// Mitsubishi GX Works2 project: FRA 451 Class Project NEW   PLC: FX3G

PROGRAM MAIN
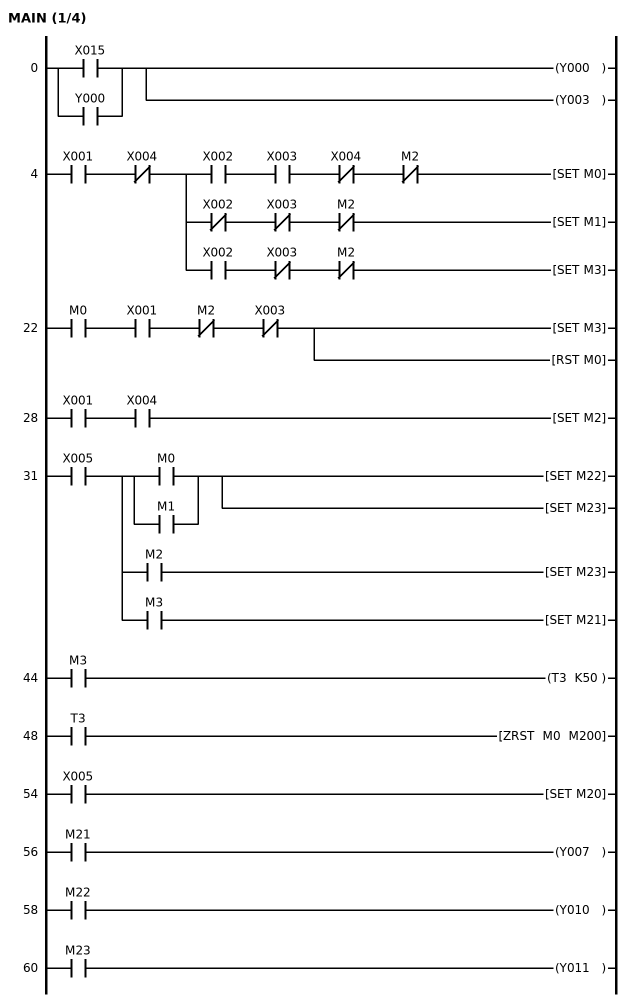
0     LD      X015
      OR      Y000
      OUT     Y000
      OUT     Y003
4     LD      X001
      ANI     X004
      MPS
      AND     X002
      AND     X003
      ANI     X004
      ANI     M2
      SET     M0
      MRD
      ANI     X002
      ANI     X003
      ANI     M2
      SET     M1
      MPP
      AND     X002
      ANI     X003
      ANI     M2
      SET     M3
22    LD      M0
      AND     X001
      ANI     M2
      ANI     X003
      SET     M3
      RST     M0
28    LD      X001
      AND     X004
      SET     M2
31    LD      X005
      MPS
      LD      M0
      OR      M1
      ANB
      SET     M22
      SET     M23
      MRD
      AND     M2
      SET     M23
      MPP
      AND     M3
      SET     M21
44    LD      M3
      OUT     T3 K50
48    LD      T3
      ZRST    M0 M200
54    LD      X005
      SET     M20
56    LD      M21
      OUT     Y007
58    LD      M22
      OUT     Y010
60    LD      M23
      OUT     Y011
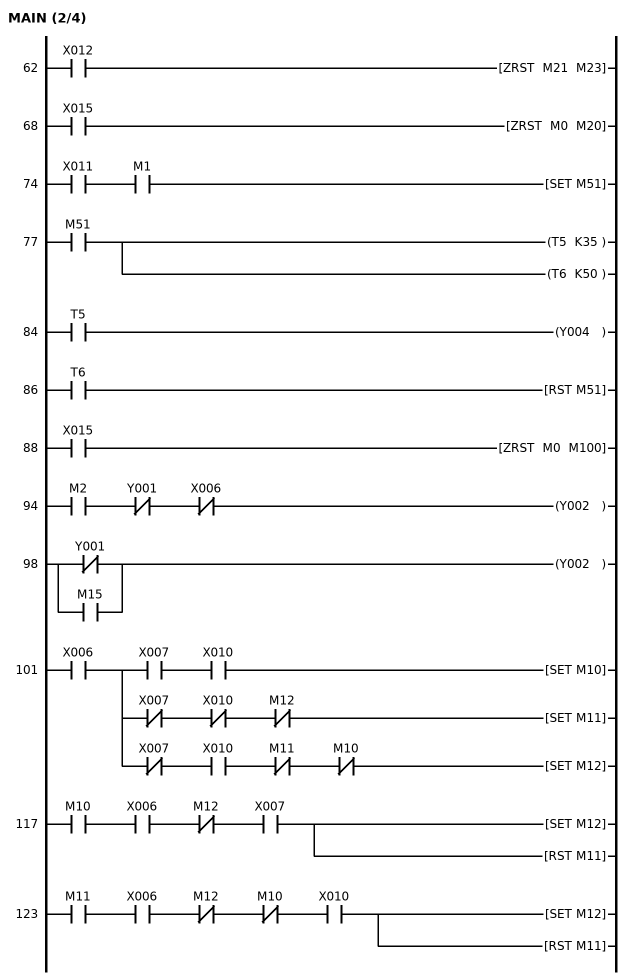
62    LD      X012
      ZRST    M21 M23
68    LD      X015
      ZRST    M0 M20
74    LD      X011
      AND     M1
      SET     M51
77    LD      M51
      OUT     T5 K35
      OUT     T6 K50
84    LD      T5
      OUT     Y004
86    LD      T6
      RST     M51
88    LD      X015
      ZRST    M0 M100
94    LD      M2
      ANI     Y001
      ANI     X006
      OUT     Y002
98    LDI     Y001
      OR      M15
      OUT     Y002
101   LD      X006
      MPS
      AND     X007
      AND     X010
      SET     M10
      MRD
      ANI     X007
      ANI     X010
      ANI     M12
      SET     M11
      MPP
      ANI     X007
      AND     X010
      ANI     M11
      ANI     M10
      SET     M12
117   LD      M10
      AND     X006
      ANI     M12
      AND     X007
      SET     M12
      RST     M11
123   LD      M11
      AND     X006
      ANI     M12
      ANI     M10
      AND     X010
      SET     M12
      RST     M11
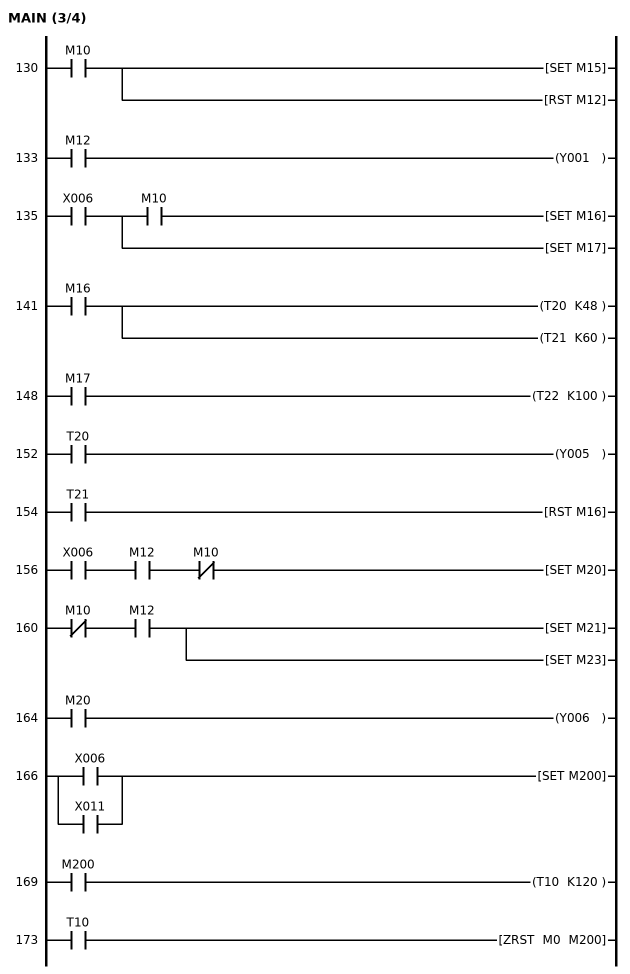
130   LD      M10
      SET     M15
      RST     M12
133   LD      M12
      OUT     Y001
135   LD      X006
      MPS
      AND     M10
      SET     M16
      MPP
      SET     M17
141   LD      M16
      OUT     T20 K48
      OUT     T21 K60
148   LD      M17
      OUT     T22 K100
152   LD      T20
      OUT     Y005
154   LD      T21
      RST     M16
156   LD      X006
      AND     M12
      ANI     M10
      SET     M20
160   LDI     M10
      AND     M12
      SET     M21
      SET     M23
164   LD      M20
      OUT     Y006
166   LD      X006
      OR      X011
      SET     M200
169   LD      M200
      OUT     T10 K120
173   LD      T10
      ZRST    M0 M200
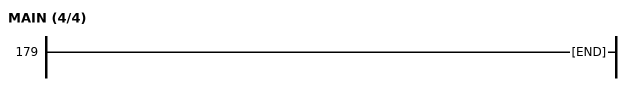
179   END
END_PROGRAM
